Fanuc KAREL source: KD00074.KL

PROGRAM KD00074
%NOLOCKGROUP
VAR
  I: INTEGER
  J: INTEGER
  B: BOOLEAN
  R: REAL
  S: STRING[80]
BEGIN
  CANCEL
END KD00074
